FUNCTION_BLOCK GenericCylinderModelType1 (* Linear motor with two position sensors and load *)
  (* Standard: 61499-2 *)
  (* Version 1.0, 2011-04-20, Sandeep Patil, The University of Auckland, First build. *)
  (* Compiler header: package fb.rt.pnp; *)
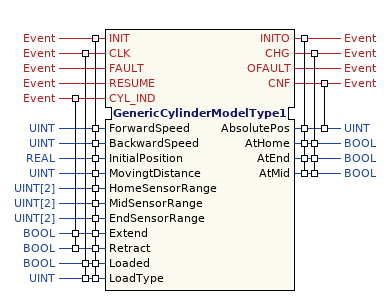
  EVENT_INPUT
    INIT WITH ForwardSpeed, BackwardSpeed, Extend, Retract, HomeSensorRange, EndSensorRange, InitialPosition, LoadType, MovingtDistance, Loaded, MidSensorRange; (* Initialization Request *)
    CLK WITH LoadType, Loaded; (* Clock signal *)
    FAULT;
    RESUME;
    CYL_IND WITH Extend, Retract;
  END_EVENT
  EVENT_OUTPUT
    INITO WITH AbsolutePos, AtHome, AtEnd, AtMid; (* Initialization Confirm *)
    CHG WITH AtEnd, AtHome, AtMid; (* Indicate data outputs changed *)
    OFAULT;
    CNF WITH AbsolutePos;
  END_EVENT
  VAR_INPUT
    ForwardSpeed : UINT; (* Forward speed *)
    BackwardSpeed : UINT; (* Backward speed *)
    InitialPosition : REAL; (* Initial position *)
    MovingtDistance : UINT; (* Moving distance *)
    HomeSensorRange : ARRAY [0..1] OF UINT; (* Detection range of home sensor *)
    MidSensorRange : ARRAY [0..1] OF UINT; (* Detection range of home sensor *)
    EndSensorRange : ARRAY [0..1] OF UINT; (* Detection range of end sensor *)
    Extend : BOOL;
    Retract : BOOL;
    Loaded : BOOL;
    LoadType : UINT;
  END_VAR
  VAR_OUTPUT
    AbsolutePos : UINT; (* Current position *)
    AtHome : BOOL; (* Detected at home position *)
    AtEnd : BOOL; (* Detected at end position *)
    AtMid : BOOL;
  END_VAR
  FBS
    Home : PnPSensor;
    Middle : PnPSensor;
    End : PnPSensor;
    MovingStatus : MovementBlockType1;
    Position : LinearMotionLoad;
  END_FBS
  EVENT_CONNECTIONS
    INIT TO MovingStatus.INIT;
    FAULT TO MovingStatus.FAULT;
    RESUME TO MovingStatus.RESUME;
    Home.CHG TO CHG;
    End.CHG TO CHG;
    End.INITO TO INITO;
    MovingStatus.OFAULT TO OFAULT;
    MovingStatus.INITO TO Position.INIT;
    Position.INITO TO Home.INIT;
    Position.CHG TO Home.CLK;
    Position.CHG TO End.CLK;
    Home.INITO TO Middle.INIT;
    Middle.INITO TO End.INIT;
    Position.CHG TO Middle.CLK;
    Position.CHG TO CNF;
    Middle.CHG TO CHG;
    CLK TO Position.CLK;
    CYL_IND TO MovingStatus.CLK;
  END_CONNECTIONS
  DATA_CONNECTIONS
    EndSensorRange TO End.Zone;
    MovingStatus.C_FWD TO Position.MoveForwards;
    MovingStatus.C_BWD TO Position.MoveBackwards;
    Loaded TO Position.Loaded;
    ForwardSpeed TO Position.ForwardSpeed;
    BackwardSpeed TO Position.BackwardSpeed;
    LoadType TO Position.LoadType;
    Position.AbsolutePos TO AbsolutePos;
    MovingtDistance TO Position.MovingDistance;
    Home.Detected TO AtHome;
    End.Detected TO AtEnd;
    InitialPosition TO Position.InitialPosition;
    HomeSensorRange TO Home.Zone;
    Position.RelativePos TO Home.Position;
    Position.RelativePos TO End.Position;
    Position.RelativePos TO Middle.Position;
    MidSensorRange TO Middle.Zone;
    Middle.Detected TO AtMid;
    Extend TO MovingStatus.Extend;
    Retract TO MovingStatus.Retract;
  END_CONNECTIONS
END_FUNCTION_BLOCK
